{attribute 'GeneratedUsingTerminal: EL2252-0000-0016'}
{attribute addProperty BoxType "EL2252-0000-0016"}
{attribute addProperty Description "EL2252 2Ch. Dig. Output 24V, 0.5A, DC Time Stamp"}
{attribute addProperty Physics "KK"}
{attribute addProperty Id "DC_Sync_ActivateAT %Q*DC_Sync_Activate_FA2D29101DC_Sync_StartAT %Q*DC_Sync_Start_E82E92338Channel_1AT %Q*Channel_42CA91F71Channel_2AT %Q*Channel_42CA91F71WcStateAT %I*WcState_0B2B16F91InfoDataAT %I*InfoData_A7436BC610"}
{attribute addProperty CRC "3172021446"}
{attribute addProperty Size "22"}
TYPE EL2252_BD1134C6 EXTENDS EtcSlaveTerminalBase_947E5A46 :
STRUCT
	{attribute addProperty Name "DC_Sync_Activate"}
	DC_Sync_Activate : DC_Sync_Activate_FA2D2910;
	{attribute addProperty Name "DC_Sync_Start"}
	DC_Sync_Start : DC_Sync_Start_E82E9233;
	{attribute addProperty Name "Channel_1"}
	Channel_1 : Channel_42CA91F7;
	{attribute addProperty Name "Channel_2"}
	Channel_2 : Channel_42CA91F7;
	{attribute addProperty Name "WcState"}
	WcState : WcState_0B2B16F9;
	{attribute addProperty Name "InfoData"}
	InfoData : InfoData_A7436BC6;
END_STRUCT
END_TYPE

(* stored: Version 1.2.0.0, ProductVersion 3.1.4024.11
   DUT EL2252_BD1134C6: Id {bab51a4b-e68d-4179-bdb5-c3d7b41c11aa} *)
